// TIA Portal project "PlcProjekt" (V17)

(* hardware
DEVICE "S7-1200-Station_1"  S7-1200 Station
   slot 0: "Baugruppenträger_0"  S7-1200 Rack  Rack  V1.0
   slot 1: "PLC_1"  CPU 1214C DC/DC/DC  6ES7 214-1AG40-0XB0  V4.2
   slot 3: "AQ 1x12BIT_1"  AQ1 signal board  6ES7 232-4HA30-0XB0  V1.0
*)

// ===== PLC "PLC_1"  CPU 1214C DC/DC/DC =====

VAR_GLOBAL   // PLC tag table "Standard-Variablentabelle"
   "System_Byte" AT %MB100 : Byte;
   "FirstScan" AT %M100.0 : Bool;
   "DiagStatusUpdate" AT %M100.1 : Bool;
   "AlwaysTRUE" AT %M100.2 : Bool;
   "AlwaysFALSE" AT %M100.3 : Bool;
   "Clock_Byte" AT %MB110 : Byte;
   "Clock_10Hz" AT %M110.0 : Bool;
   "Clock_5Hz" AT %M110.1 : Bool;
   "Clock_2.5Hz" AT %M110.2 : Bool;
   "Clock_2Hz" AT %M110.3 : Bool;
   "Clock_1.25Hz" AT %M110.4 : Bool;
   "Clock_1Hz" AT %M110.5 : Bool;
   "Clock_0.625Hz" AT %M110.6 : Bool;
   "Clock_0.5Hz" AT %M110.7 : Bool;
   "S1" AT %I0.0 : Bool;   // Taster Start
   "P1" AT %Q0.0 : Bool;   // Meldeleuchte
END_VAR

DATA_BLOCK "PcToPlc"   // DB1
{ S7_Optimized_Access := 'FALSE' }
VERSION : 0.1
   VAR
      Plc : Array[0..256] of Byte;
   END_VAR
BEGIN
END_DATA_BLOCK

DATA_BLOCK "PlcToPc"   // DB2
{ S7_Optimized_Access := 'FALSE' }
VERSION : 0.1
   VAR
      Plc : Array[0..256] of Byte;
   END_VAR
BEGIN
END_DATA_BLOCK

DATA_BLOCK "DeleteMe_DB"   // DB3
{ S7_Optimized_Access := 'TRUE' }
VERSION : 0.1
// stored: InstanceOfName DeleteMe
"DeleteMe"
BEGIN
END_DATA_BLOCK

FUNCTION_BLOCK "DeleteMe"   // FB1, SCL
{ S7_Optimized_Access := 'TRUE' }
VERSION : 0.1
   VAR
      Eingeschaltet : Bool;
      Gesamtzeit : TON_TIME;
   END_VAR
BEGIN
END_FUNCTION_BLOCK

FUNCTION "DatenRangieren" : Void   // FC1, SCL
{ S7_Optimized_Access := 'TRUE' }
VERSION : 0.1
   VAR_TEMP
      TextLaenge : UInt;
   END_VAR
BEGIN
   // Area 16#81 --> Input
   // Area 16#82 --> Output
   // Area 16#84 --> DB

   IF  "PcToPlc".Plc[96].%X0 THEN
       // Simulation aktiv --> DI werden vom PC überschrieben
       POKE(area := 16#81,                     // DI (Hardware PLC)
           dbNumber := 0,
           byteOffset := 0,
           value := PEEK(area := 16#84, dbNumber := 1, byteOffset := 0));
   ELSE
       // Hardware aktiv --> DI werden zum PC übertragen
       POKE(area := 16#84,                    // Datenbausteine
           dbNumber := 1,                     // DB1 -> Pc2Plc
           byteOffset := 0,                   // Byte 0
           value := PEEK(area := 16#81, dbNumber := 0, byteOffset := 0));
   END_IF;

   // DQ werden immer zum PC übertragen
   POKE(area := 16#84,                         // Datenbausteine
        dbNumber := 2,                         // DB1 -> Pc2Plc
        byteOffset := 0,
        value := PEEK(area := 16#82, dbNumber := 0, byteOffset := 0));

   Strg_TO_Chars(Strg := 'Fibonacci V3.0',
                 pChars := 96,
                 Cnt=>#TextLaenge,
                 Chars := "PlcToPc".Plc);
END_FUNCTION

ORGANIZATION_BLOCK "Main"   // OB1, LAD, ProgramCycle
TITLE = "Main Program Sweep (Cycle)"
{ S7_Optimized_Access := 'TRUE' }
VERSION : 0.1
   VAR_INPUT
      Initial_Call : Bool;   // Initial call of this OB
      Remanence : Bool;   // =True, if remanent data are available
   END_VAR
BEGIN

REGION Network 1
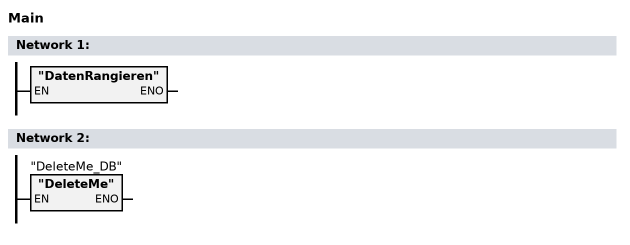
   RUNG wire#powerrail
      "DatenRangieren"()
   END_RUNG
   // the same network as SCL:
   "DatenRangieren"();
END_REGION

REGION Network 2
   RUNG wire#powerrail
      "DeleteMe_DB"()
   END_RUNG
   // the same network as SCL:
   "DeleteMe_DB"();   // "DeleteMe"
END_REGION
END_ORGANIZATION_BLOCK

ORGANIZATION_BLOCK "Startup"   // OB100, SCL, Startup
TITLE = "Complete Restart"
{ S7_Optimized_Access := 'TRUE' }
VERSION : 0.1
   VAR_INPUT
      LostRetentive : Bool;   // True if retentive data are lost
      LostRTC : Bool;   // True if date and time are lost
   END_VAR
BEGIN
   // Area 16#81 --> Input
   // Area 16#82 --> Output
   // Area 16#84 --> DB

   POKE(area := 16#82, dbNumber := 0, byteOffset := 0, value := byte#0);  // Ausgänge löschen
END_ORGANIZATION_BLOCK